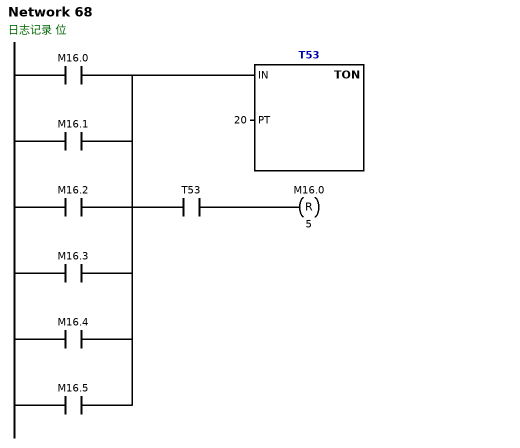
[picture p24: OB1 networks 68-68]
Network 68
// 日志记录 位
LD     M16.0
O      M16.1
O      M16.2
O      M16.3
O      M16.4
O      M16.5
TON    T53, 20
A      T53
R      M16.0, 5
END_ORGANIZATION_BLOCK

SUBROUTINE_BLOCK M进样下:SBR0
TITLE=子程序注释
VAR_INPUT
次数:WORD;	// LW0 
报警T:WORD;	// LW2 
反推T:WORD;	// LW4 
END_VAR
VAR_IN_OUT
启动位:BOOL;	// L6.0 
END_VAR
VAR_OUTPUT
结束位:BOOL;	// L6.1 
采样阀:BOOL;	// L6.2 
alarm:BOOL;	// L6.3 
END_VAR
BEGIN
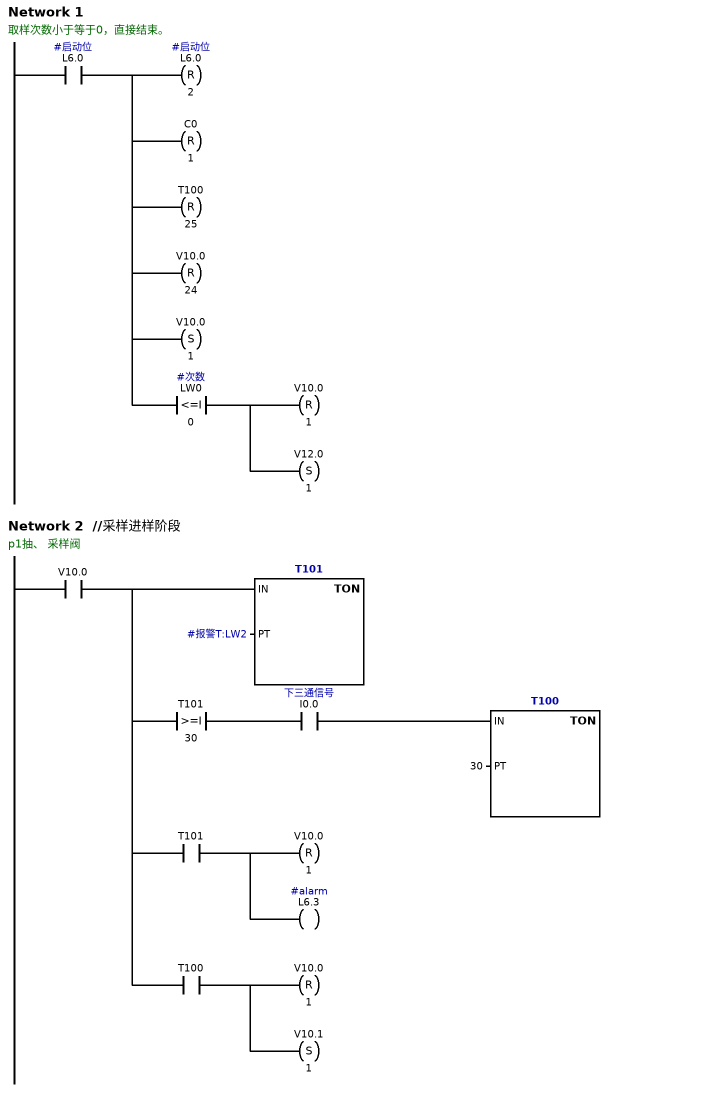
Network 1
// 取样次数小于等于0，直接结束。
LD     #启动位:L6.0
R      #启动位:L6.0, 2
R      C0, 1
R      T100, 25
R      V10.0, 24
S      V10.0, 1
AW<=   #次数:LW0, 0
R      V10.0, 1
S      V12.0, 1
Network 2 // //采样进样阶段
// p1抽、 采样阀
LD     V10.0
LPS
TON    T101, #报警T:LW2
AW>=   T101, 30
A      下三通信号:I0.0
TON    T100, 30
LRD
A      T101
R      V10.0, 1
=      #alarm:L6.3
LPP
A      T100
R      V10.0, 1
S      V10.1, 1
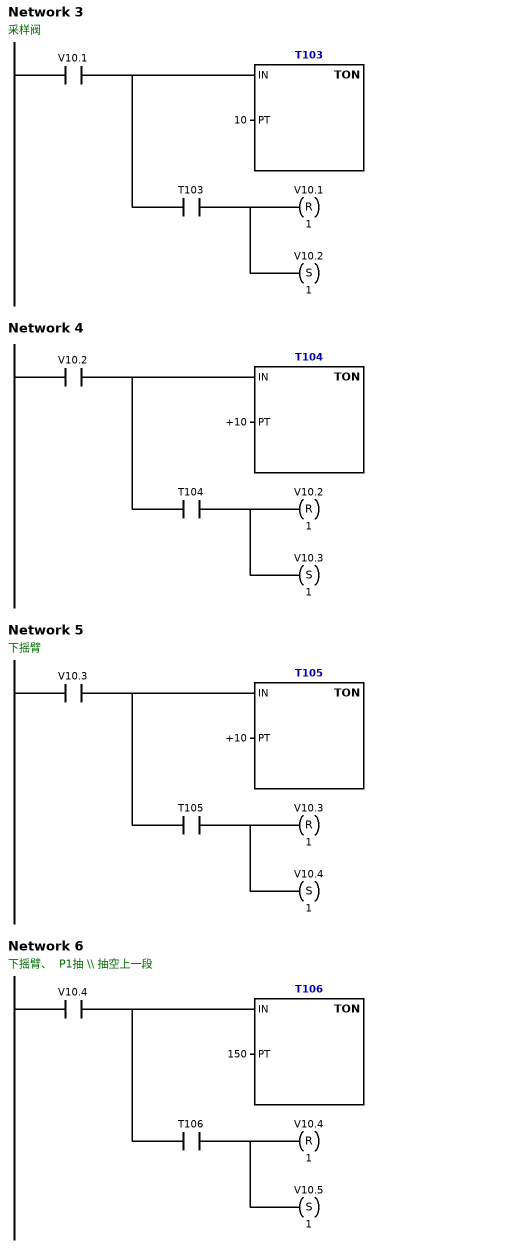
Network 3
// 采样阀  
LD     V10.1
TON    T103, 10
A      T103
R      V10.1, 1
S      V10.2, 1
Network 4
LD     V10.2
TON    T104, +10
A      T104
R      V10.2, 1
S      V10.3, 1
Network 5
// 下摇臂
LD     V10.3
TON    T105, +10
A      T105
R      V10.3, 1
S      V10.4, 1
Network 6
//  下摇臂、  P1抽 \\ 抽空上一段
LD     V10.4
TON    T106, 150
A      T106
R      V10.4, 1
S      V10.5, 1
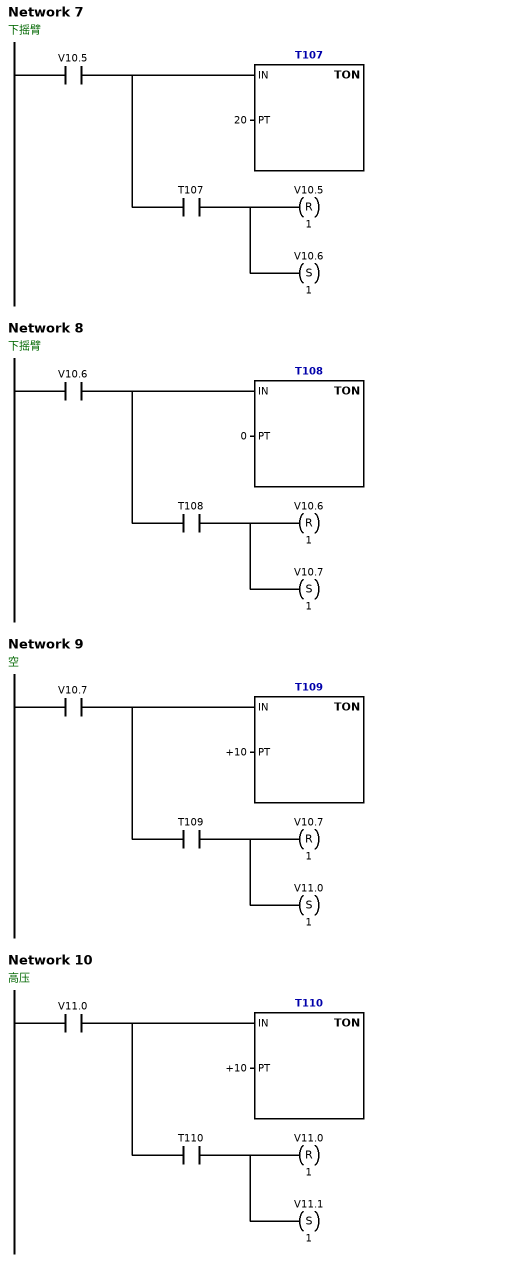
Network 7
//  下摇臂   
LD     V10.5
TON    T107, 20
A      T107
R      V10.5, 1
S      V10.6, 1
Network 8
// 下摇臂
LD     V10.6
TON    T108, 0
A      T108
R      V10.6, 1
S      V10.7, 1
Network 9
// 空
LD     V10.7
TON    T109, +10
A      T109
R      V10.7, 1
S      V11.0, 1
Network 10
// 高压
LD     V11.0
TON    T110, +10
A      T110
R      V11.0, 1
S      V11.1, 1
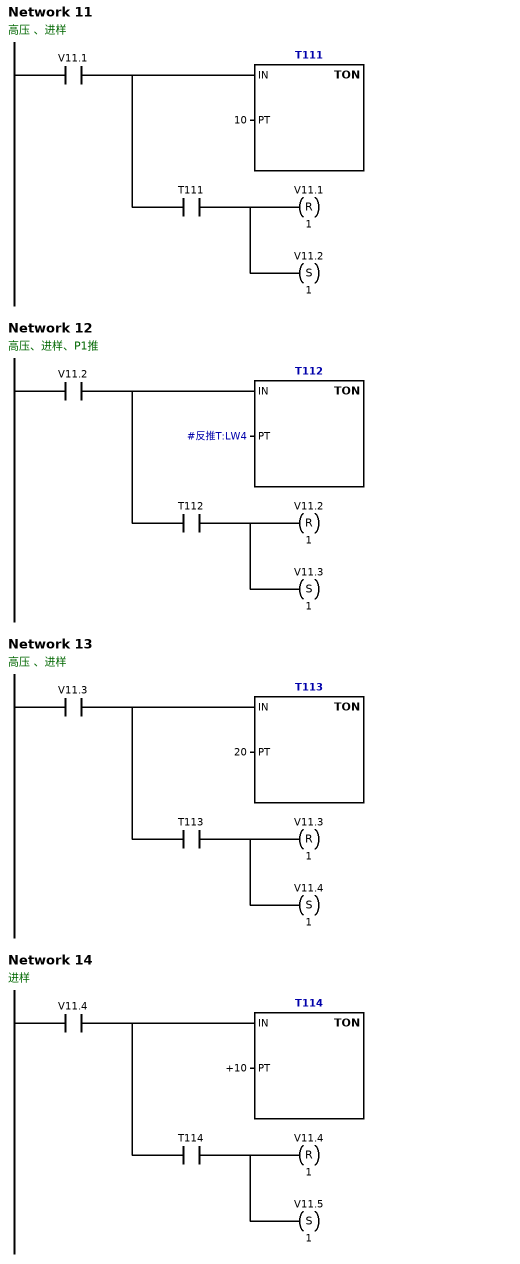
Network 11
// 高压 、进样
LD     V11.1
TON    T111, 10
A      T111
R      V11.1, 1
S      V11.2, 1
Network 12
// 高压、进样、P1推
LD     V11.2
TON    T112, #反推T:LW4
A      T112
R      V11.2, 1
S      V11.3, 1
Network 13
// 高压 、进样
LD     V11.3
TON    T113, 20
A      T113
R      V11.3, 1
S      V11.4, 1
Network 14
// 进样
LD     V11.4
TON    T114, +10
A      T114
R      V11.4, 1
S      V11.5, 1
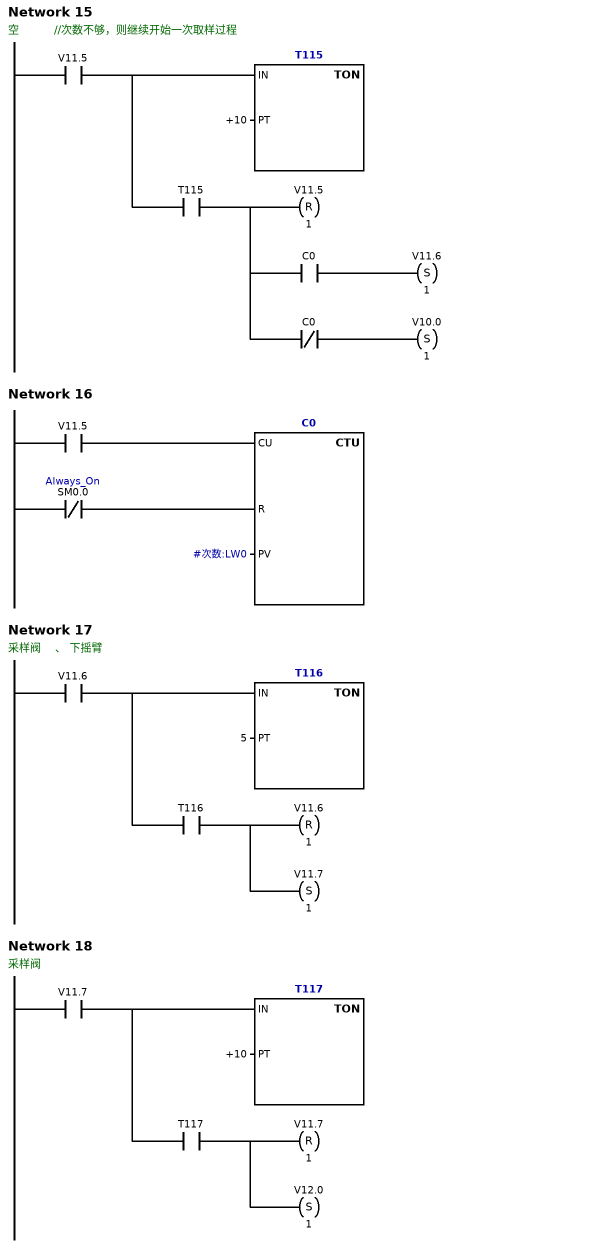
Network 15
// 空          //次数不够，则继续开始一次取样过程
LD     V11.5
TON    T115, +10
A      T115
LPS
R      V11.5, 1
A      C0
S      V11.6, 1
LPP
AN     C0
S      V10.0, 1
Network 16
LD     V11.5
LDN    Always_On:SM0.0
CTU    C0, #次数:LW0
Network 17
// 采样阀    、 下摇臂
LD     V11.6
TON    T116, 5
A      T116
R      V11.6, 1
S      V11.7, 1
Network 18
// 采样阀 
LD     V11.7
TON    T117, +10
A      T117
R      V11.7, 1
S      V12.0, 1
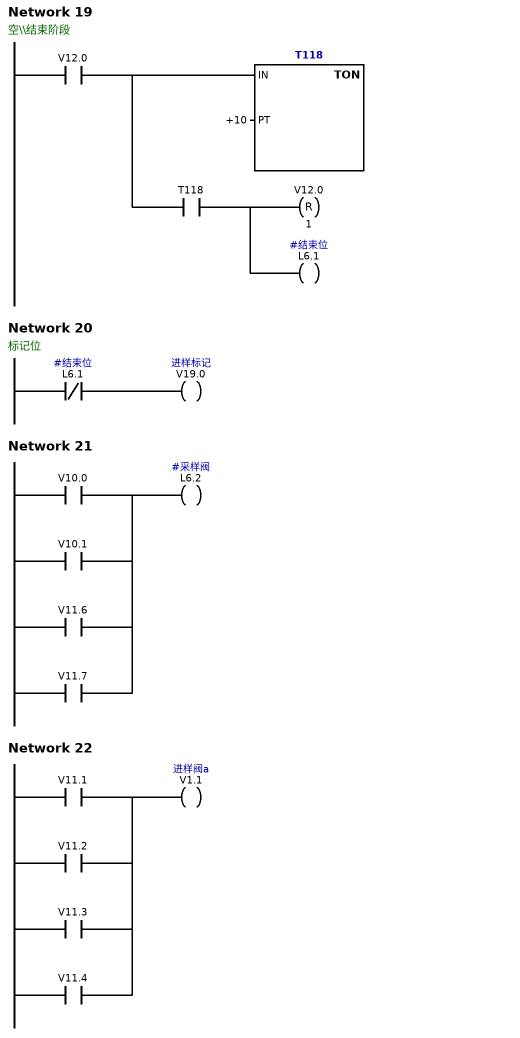
Network 19
// 空\\结束阶段
LD     V12.0
TON    T118, +10
A      T118
R      V12.0, 1
=      #结束位:L6.1
Network 20
// 标记位
LDN    #结束位:L6.1
=      进样标记:V19.0
Network 21
LD     V10.0
O      V10.1
O      V11.6
O      V11.7
=      #采样阀:L6.2
Network 22
LD     V11.1
O      V11.2
O      V11.3
O      V11.4
=      进样阀a:V1.1
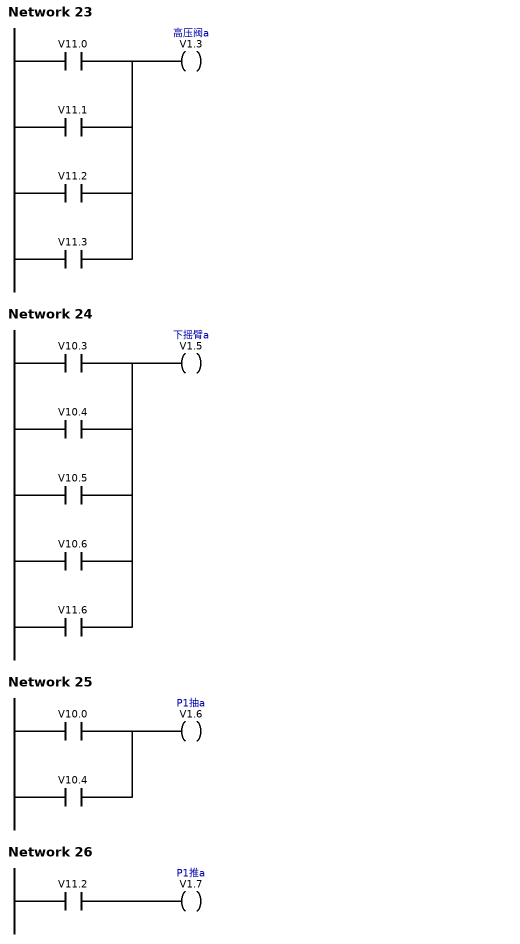
Network 23
LD     V11.0
O      V11.1
O      V11.2
O      V11.3
=      高压阀a:V1.3
Network 24
LD     V10.3
O      V10.4
O      V10.5
O      V10.6
O      V11.6
=      下摇臂a:V1.5
Network 25
LD     V10.0
O      V10.4
=      P1抽a:V1.6
Network 26
LD     V11.2
=      P1推a:V1.7
Network 28 // 网络标题
// 网络注释
END_SUBROUTINE_BLOCK

SUBROUTINE_BLOCK M进样简:SBR1
TITLE=
VAR_INPUT
次数:WORD;	// LW0 
报警T:WORD;	// LW2 
反推T:WORD;	// LW4 
信号:BOOL;	// L6.0 
END_VAR
VAR_IN_OUT
启动位:BOOL;	// L6.1 
END_VAR
VAR_OUTPUT
结束位:BOOL;	// L6.2 
采样阀:BOOL;	// L6.3 
alarm:BOOL;	// L6.4 
END_VAR
BEGIN
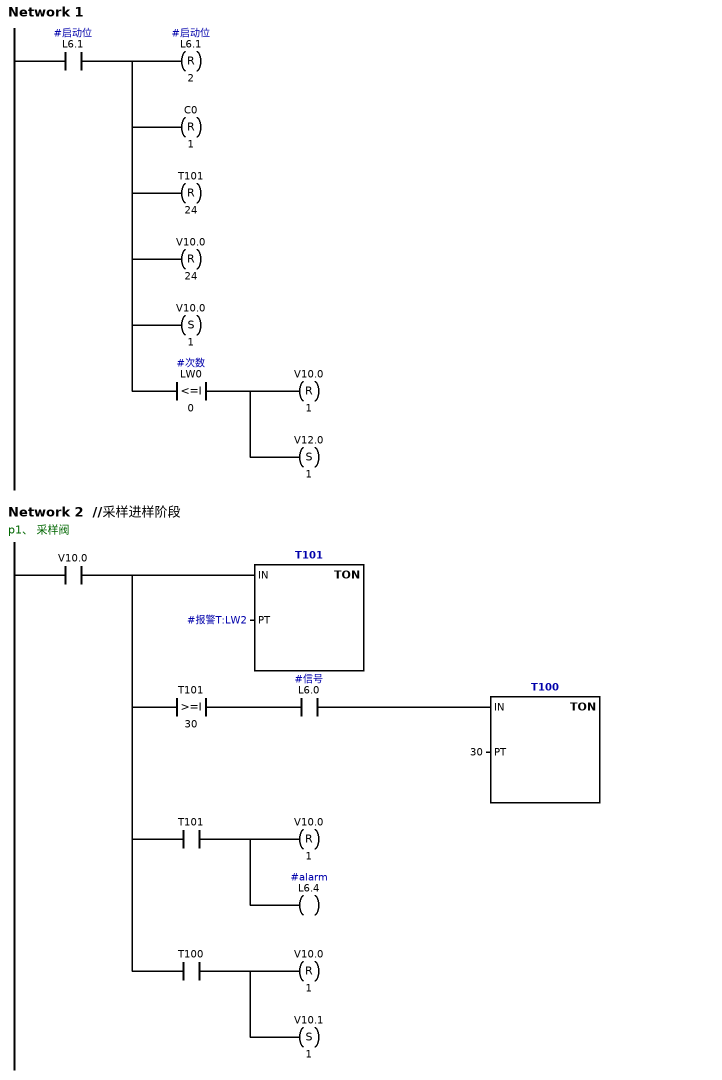
Network 1
LD     #启动位:L6.1
R      #启动位:L6.1, 2
R      C0, 1
R      T101, 24
R      V10.0, 24
S      V10.0, 1
AW<=   #次数:LW0, 0
R      V10.0, 1
S      V12.0, 1
Network 2 // //采样进样阶段
// p1、 采样阀 
LD     V10.0
LPS
TON    T101, #报警T:LW2
AW>=   T101, 30
A      #信号:L6.0
TON    T100, 30
LRD
A      T101
R      V10.0, 1
=      #alarm:L6.4
LPP
A      T100
R      V10.0, 1
S      V10.1, 1
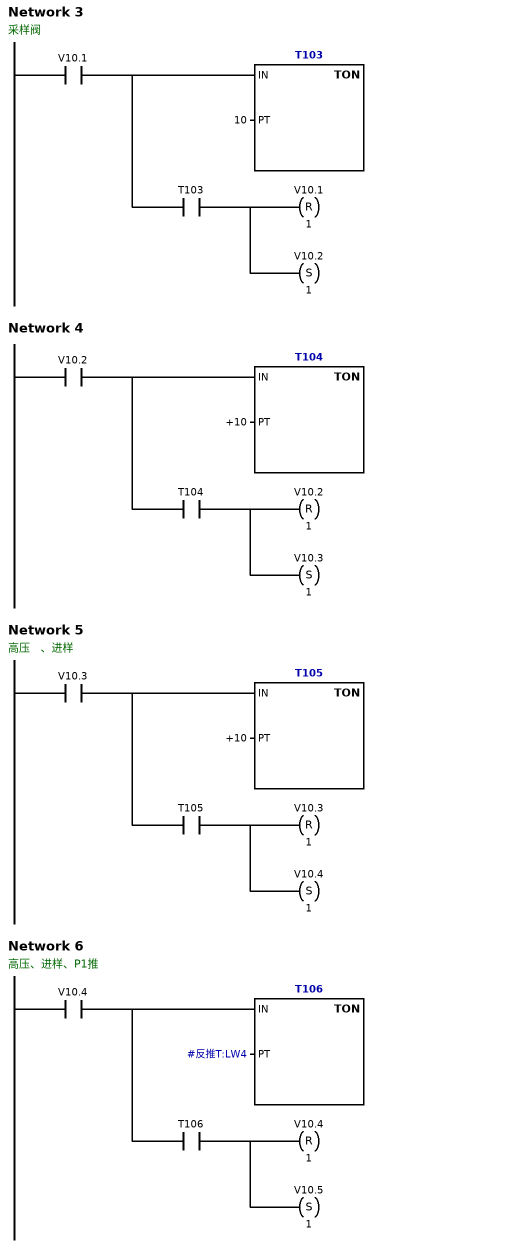
Network 3
// 采样阀  
LD     V10.1
TON    T103, 10
A      T103
R      V10.1, 1
S      V10.2, 1
Network 4
LD     V10.2
TON    T104, +10
A      T104
R      V10.2, 1
S      V10.3, 1
Network 5
// 高压   、进样
LD     V10.3
TON    T105, +10
A      T105
R      V10.3, 1
S      V10.4, 1
Network 6
// 高压、进样、P1推
LD     V10.4
TON    T106, #反推T:LW4
A      T106
R      V10.4, 1
S      V10.5, 1
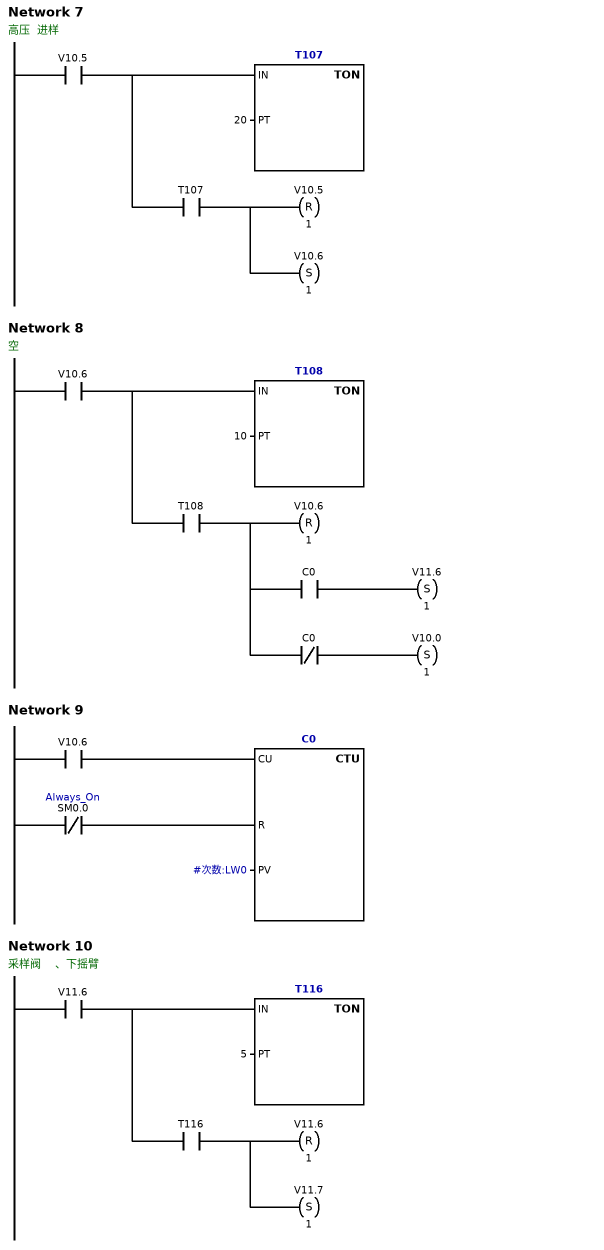
Network 7
// 高压  进样 
LD     V10.5
TON    T107, 20
A      T107
R      V10.5, 1
S      V10.6, 1
Network 8
// 空
LD     V10.6
TON    T108, 10
A      T108
LPS
R      V10.6, 1
A      C0
S      V11.6, 1
LPP
AN     C0
S      V10.0, 1
Network 9
LD     V10.6
LDN    Always_On:SM0.0
CTU    C0, #次数:LW0
Network 10
// 采样阀    、下摇臂
LD     V11.6
TON    T116, 5
A      T116
R      V11.6, 1
S      V11.7, 1
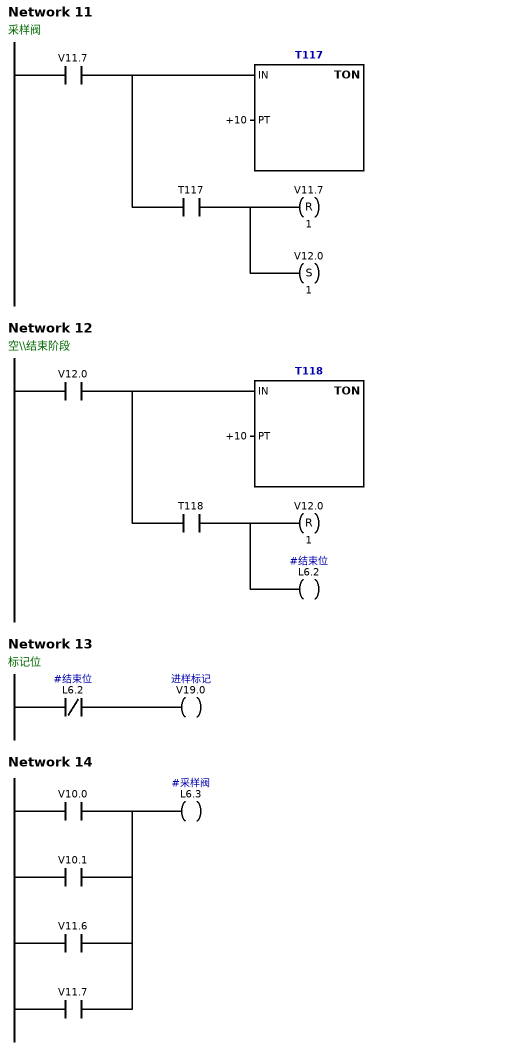
Network 11
// 采样阀 
LD     V11.7
TON    T117, +10
A      T117
R      V11.7, 1
S      V12.0, 1
Network 12
// 空\\结束阶段
LD     V12.0
TON    T118, +10
A      T118
R      V12.0, 1
=      #结束位:L6.2
Network 13
// 标记位
LDN    #结束位:L6.2
=      进样标记:V19.0
Network 14
LD     V10.0
O      V10.1
O      V11.6
O      V11.7
=      #采样阀:L6.3
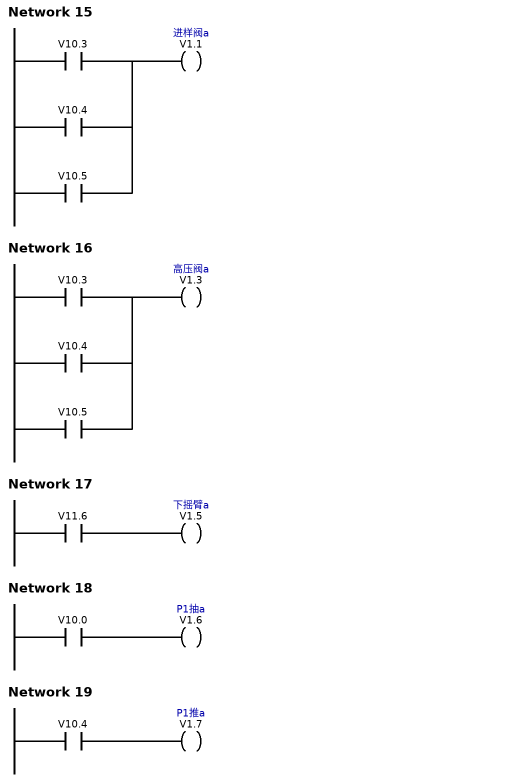
Network 15
LD     V10.3
O      V10.4
O      V10.5
=      进样阀a:V1.1
Network 16
LD     V10.3
O      V10.4
O      V10.5
=      高压阀a:V1.3
Network 17
LD     V11.6
=      下摇臂a:V1.5
Network 18
LD     V10.0
=      P1抽a:V1.6
Network 19
LD     V10.4
=      P1推a:V1.7
Network 21 // 网络标题
// 网络注释
END_SUBROUTINE_BLOCK

// SBR2: protected block, not included

SUBROUTINE_BLOCK M进硫酸:SBR3
TITLE=
VAR_INPUT
次数:WORD;	// LW0 
报警T:WORD;	// LW2 
END_VAR
VAR_IN_OUT
启动位:BOOL;	// L4.0 
END_VAR
VAR_OUTPUT
结束位:BOOL;	// L4.1 
采样阀:BOOL;	// L4.2 
alarm:BOOL;	// L4.3 
END_VAR
BEGIN
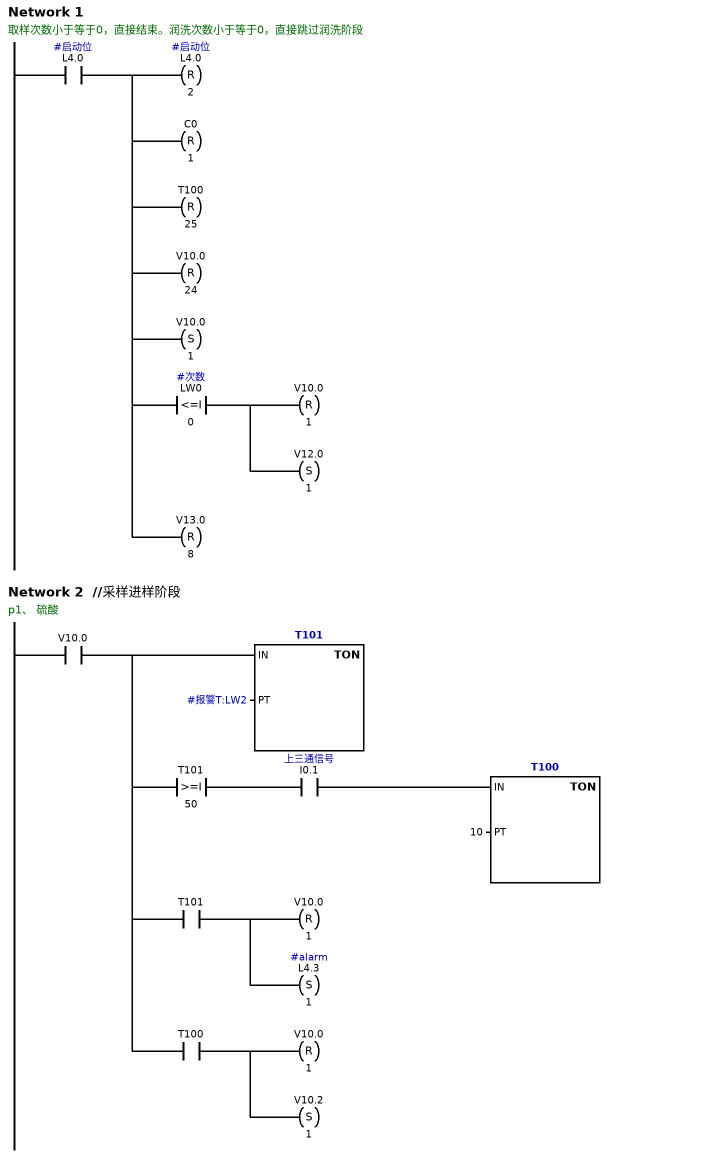
Network 1
// 取样次数小于等于0，直接结束。润洗次数小于等于0，直接跳过润洗阶段
LD     #启动位:L4.0
LPS
R      #启动位:L4.0, 2
R      C0, 1
R      T100, 25
R      V10.0, 24
S      V10.0, 1
AW<=   #次数:LW0, 0
R      V10.0, 1
S      V12.0, 1
LPP
R      V13.0, 8
Network 2 // //采样进样阶段
// p1、 硫酸
LD     V10.0
LPS
TON    T101, #报警T:LW2
AW>=   T101, 50
A      上三通信号:I0.1
TON    T100, 10
LRD
A      T101
R      V10.0, 1
S      #alarm:L4.3, 1
LPP
A      T100
R      V10.0, 1
S      V10.2, 1
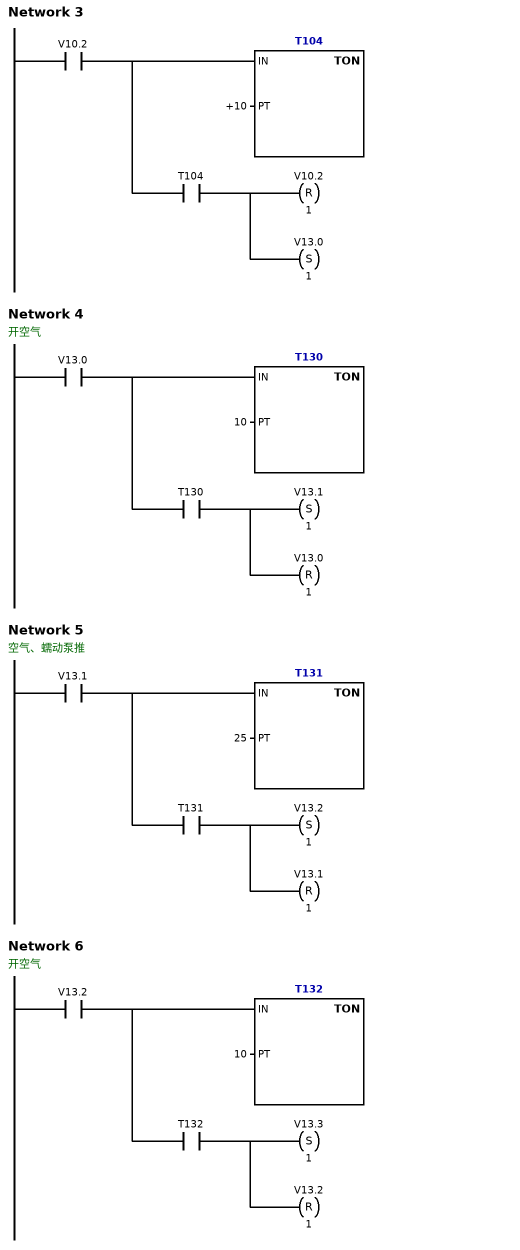
Network 3
LD     V10.2
TON    T104, +10
A      T104
R      V10.2, 1
S      V13.0, 1
Network 4
// 开空气
LD     V13.0
TON    T130, 10
A      T130
S      V13.1, 1
R      V13.0, 1
Network 5
// 空气、蠕动泵推
LD     V13.1
TON    T131, 25
A      T131
S      V13.2, 1
R      V13.1, 1
Network 6
// 开空气
LD     V13.2
TON    T132, 10
A      T132
S      V13.3, 1
R      V13.2, 1
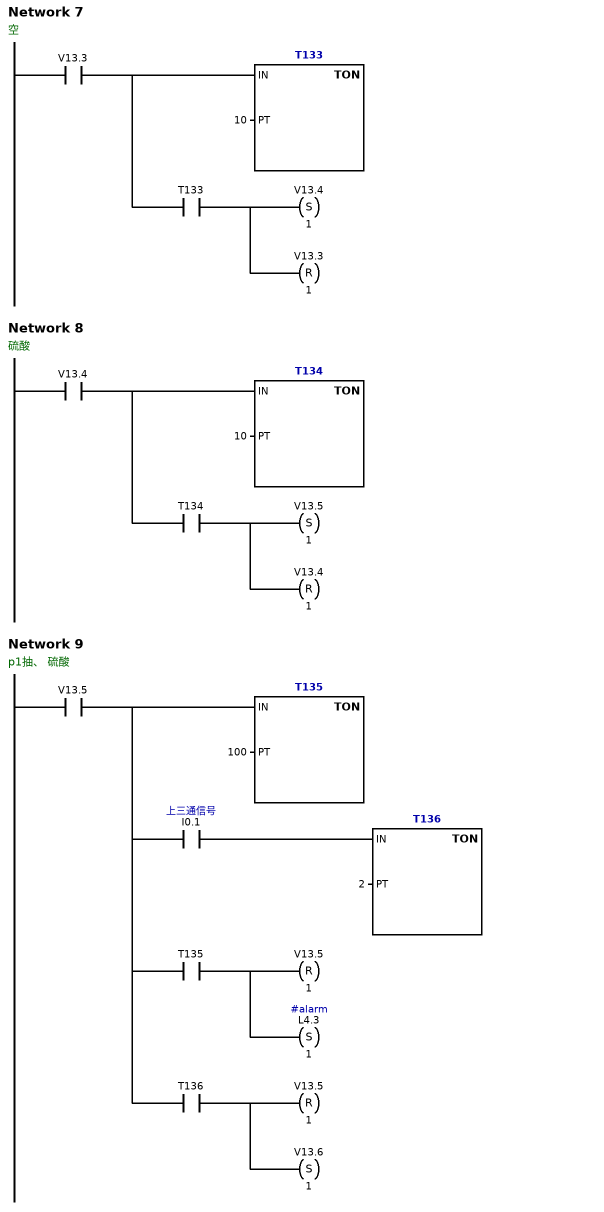
Network 7
// 空
LD     V13.3
TON    T133, 10
A      T133
S      V13.4, 1
R      V13.3, 1
Network 8
// 硫酸
LD     V13.4
TON    T134, 10
A      T134
S      V13.5, 1
R      V13.4, 1
Network 9
// p1抽、 硫酸
LD     V13.5
LPS
TON    T135, 100
A      上三通信号:I0.1
TON    T136, 2
LRD
A      T135
R      V13.5, 1
S      #alarm:L4.3, 1
LPP
A      T136
R      V13.5, 1
S      V13.6, 1
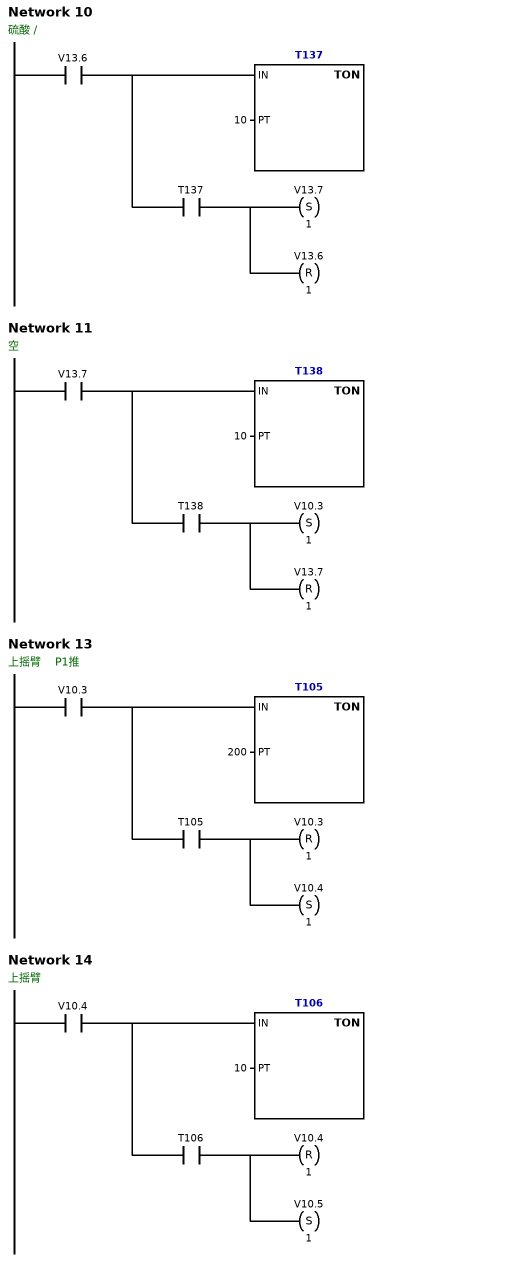
Network 10
// 硫酸
// 
LD     V13.6
TON    T137, 10
A      T137
S      V13.7, 1
R      V13.6, 1
Network 11
// 空
LD     V13.7
TON    T138, 10
A      T138
S      V10.3, 1
R      V13.7, 1
Network 13
// 上摇臂    P1推
LD     V10.3
TON    T105, 200
A      T105
R      V10.3, 1
S      V10.4, 1
Network 14
// 上摇臂
LD     V10.4
TON    T106, 10
A      T106
R      V10.4, 1
S      V10.5, 1
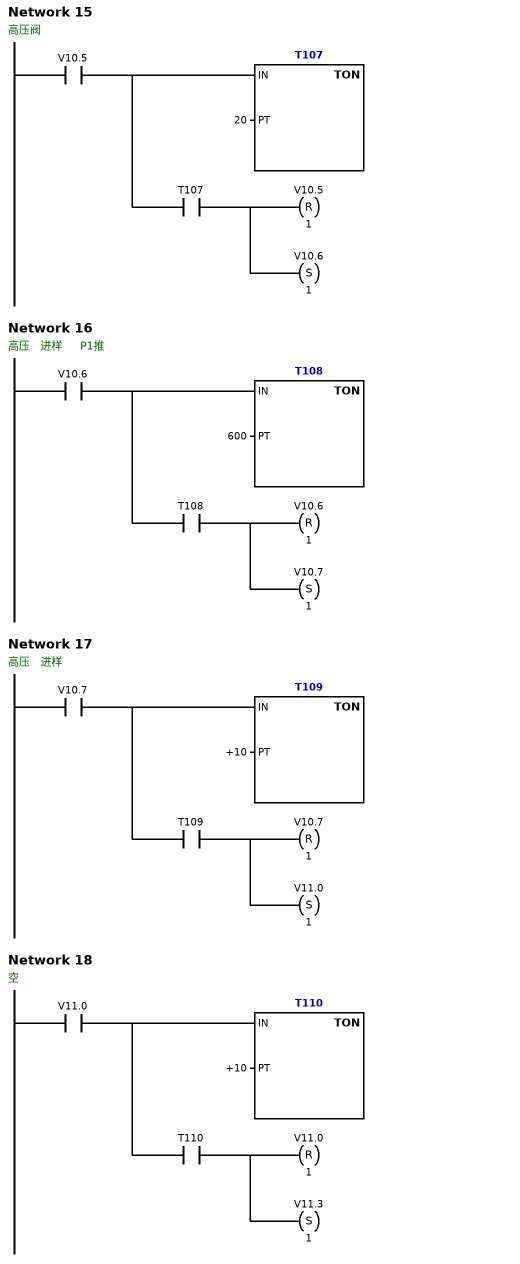
Network 15
// 高压阀
LD     V10.5
TON    T107, 20
A      T107
R      V10.5, 1
S      V10.6, 1
Network 16
// 高压   进样     P1推
LD     V10.6
TON    T108, 600
A      T108
R      V10.6, 1
S      V10.7, 1
Network 17
// 高压   进样  
LD     V10.7
TON    T109, +10
A      T109
R      V10.7, 1
S      V11.0, 1
Network 18
// 空
LD     V11.0
TON    T110, +10
A      T110
R      V11.0, 1
S      V11.3, 1
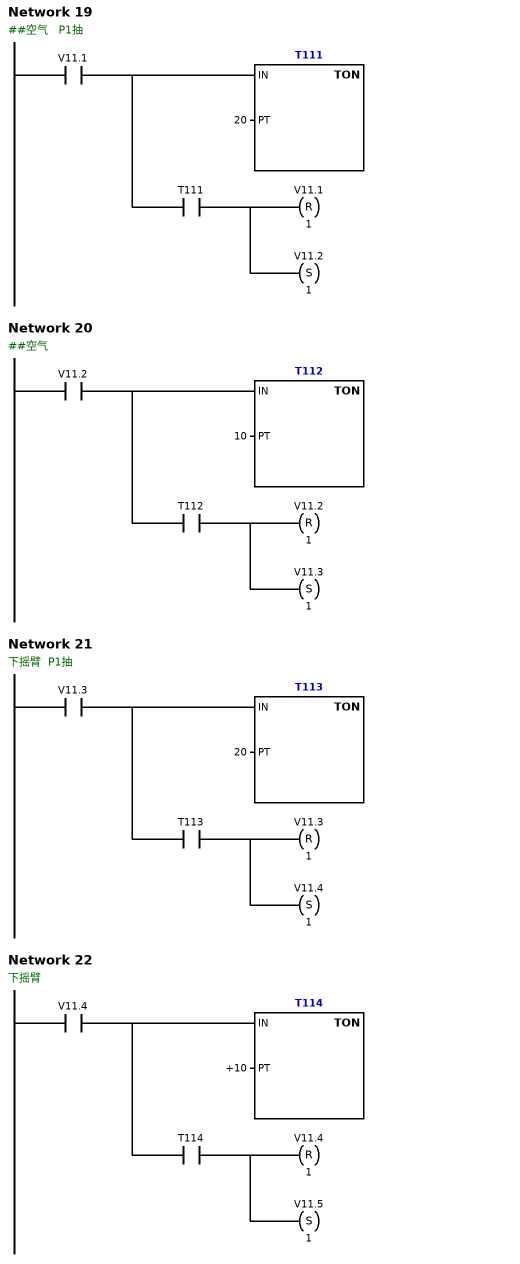
Network 19
// ##空气   P1抽
LD     V11.1
TON    T111, 20
A      T111
R      V11.1, 1
S      V11.2, 1
Network 20
// ##空气
LD     V11.2
TON    T112, 10
A      T112
R      V11.2, 1
S      V11.3, 1
Network 21
// 下摇臂  P1抽
LD     V11.3
TON    T113, 20
A      T113
R      V11.3, 1
S      V11.4, 1
Network 22
// 下摇臂
LD     V11.4
TON    T114, +10
A      T114
R      V11.4, 1
S      V11.5, 1
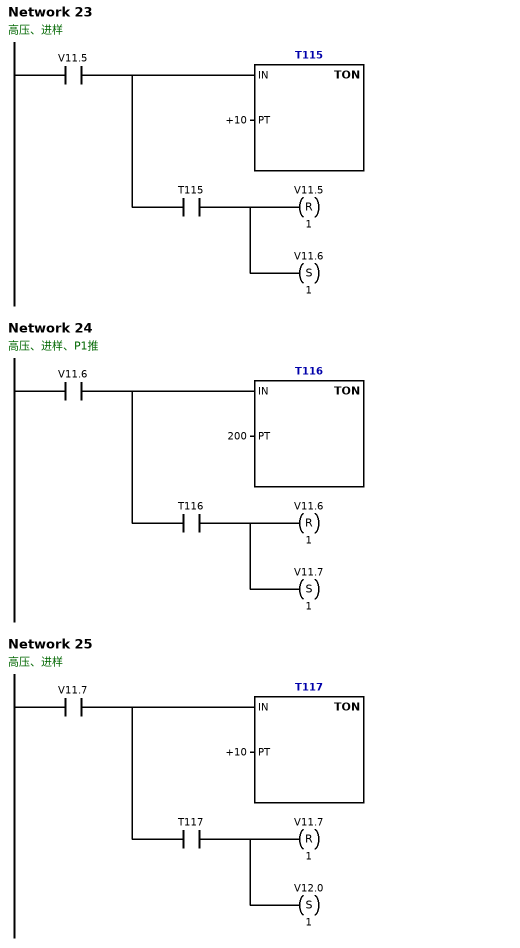
Network 23
// 高压、进样
LD     V11.5
TON    T115, +10
A      T115
R      V11.5, 1
S      V11.6, 1
Network 24
// 高压、进样、P1推  
LD     V11.6
TON    T116, 200
A      T116
R      V11.6, 1
S      V11.7, 1
Network 25
// 高压、进样
LD     V11.7
TON    T117, +10
A      T117
R      V11.7, 1
S      V12.0, 1
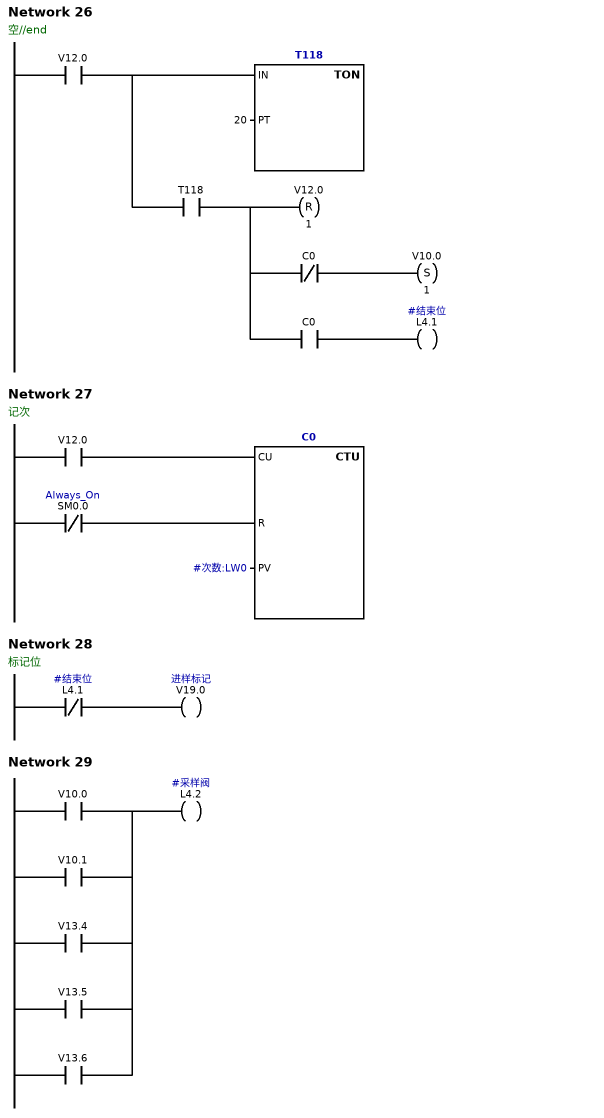
Network 26
// 空//end
LD     V12.0
TON    T118, 20
A      T118
LPS
R      V12.0, 1
AN     C0
S      V10.0, 1
LPP
A      C0
=      #结束位:L4.1
Network 27
// 记次
LD     V12.0
LDN    Always_On:SM0.0
CTU    C0, #次数:LW0
Network 28
// 标记位
LDN    #结束位:L4.1
=      进样标记:V19.0
Network 29
LD     V10.0
O      V10.1
O      V13.4
O      V13.5
O      V13.6
=      #采样阀:L4.2
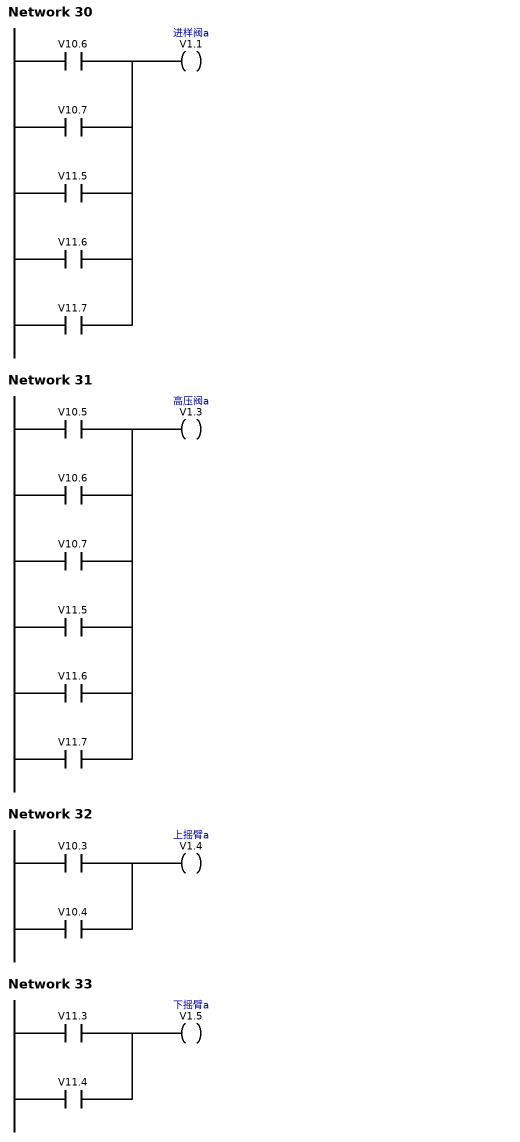
Network 30
LD     V10.6
O      V10.7
O      V11.5
O      V11.6
O      V11.7
=      进样阀a:V1.1
Network 31
LD     V10.5
O      V10.6
O      V10.7
O      V11.5
O      V11.6
O      V11.7
=      高压阀a:V1.3
Network 32
LD     V10.3
O      V10.4
=      上摇臂a:V1.4
Network 33
LD     V11.3
O      V11.4
=      下摇臂a:V1.5
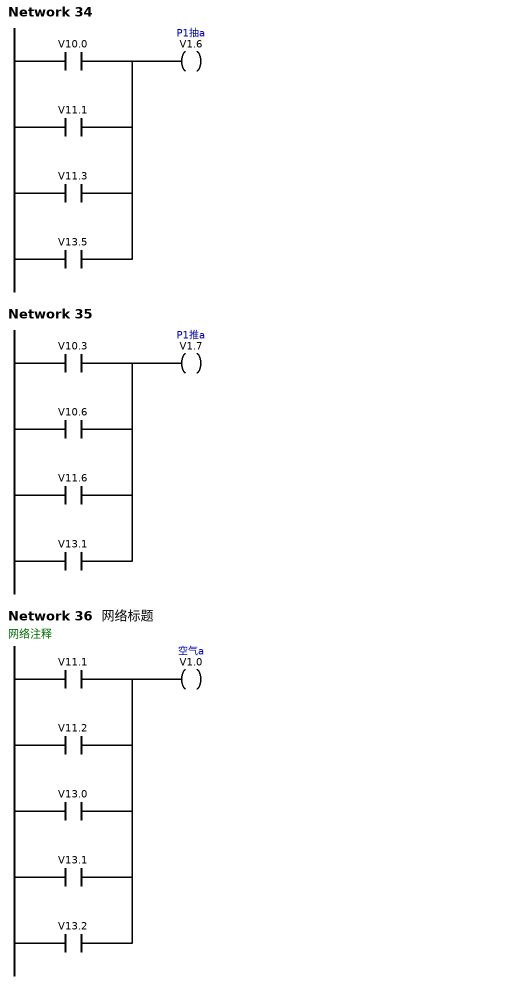
Network 34
LD     V10.0
O      V11.1
O      V11.3
O      V13.5
=      P1抽a:V1.6
Network 35
LD     V10.3
O      V10.6
O      V11.6
O      V13.1
=      P1推a:V1.7
Network 36 // 网络标题
// 网络注释
LD     V11.1
O      V11.2
O      V13.0
O      V13.1
O      V13.2
=      空气a:V1.0
END_SUBROUTINE_BLOCK

SUBROUTINE_BLOCK M去残留:SBR4
TITLE=
VAR_IN_OUT
启动位:BOOL;	// L0.0 
END_VAR
VAR_OUTPUT
结束位:BOOL;	// L0.1 
END_VAR
BEGIN
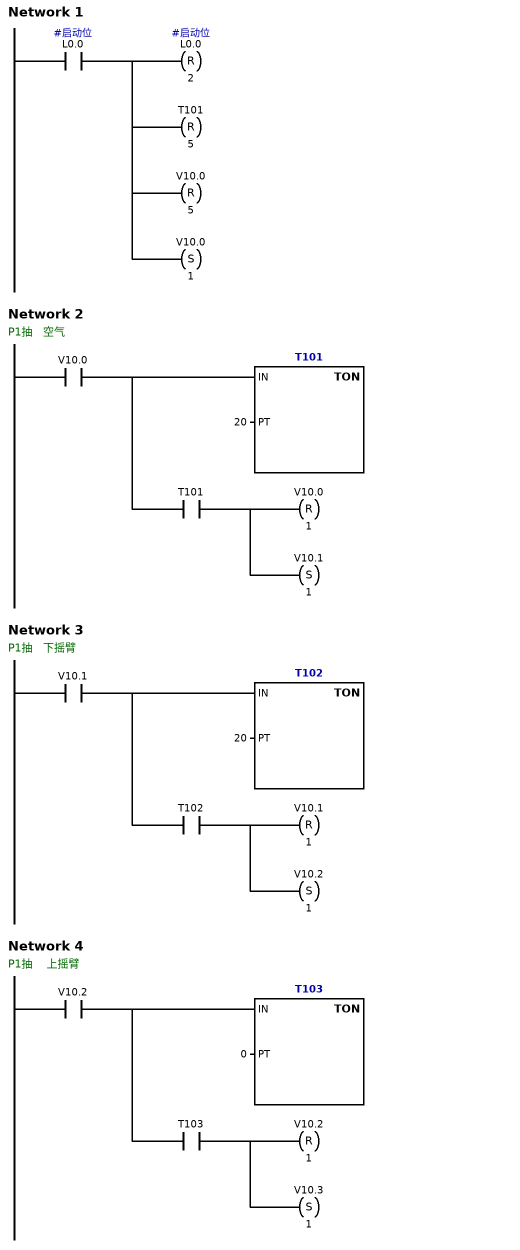
Network 1
LD     #启动位:L0.0
R      #启动位:L0.0, 2
R      T101, 5
R      V10.0, 5
S      V10.0, 1
Network 2
// P1抽   空气
LD     V10.0
TON    T101, 20
A      T101
R      V10.0, 1
S      V10.1, 1
Network 3
// P1抽   下摇臂
LD     V10.1
TON    T102, 20
A      T102
R      V10.1, 1
S      V10.2, 1
Network 4
// P1抽    上摇臂
LD     V10.2
TON    T103, 0
A      T103
R      V10.2, 1
S      V10.3, 1
